// Block: Area01_Messages

DATA_BLOCK Area01_Messages
VERSION : 0.1
   NON_RETAIN
   VAR
      A : Struct
         Msg : Array[1..352] of Bool;
         Hmi : Array[1..22] of Word;
         Ack : Array[1..22] of Word;
      END_STRUCT;
      W : Struct
         Msg : Array[1..384] of Bool;
         Hmi : Array[1..24] of Word;
         Ack : Array[1..24] of Word;
      END_STRUCT;
   END_VAR

BEGIN
   // No initialization required
END_DATA_BLOCK
